{attribute 'qualified_only'}
VAR_GLOBAL
    
	MotorPosition  		AT %I* : UINT;
	CounterOverflow 	AT %I* : BOOL;
	CounterUnderflow 	AT %I* : BOOL;
	MotorEnable			AT %Q* : BOOL;
	MotorVelocity 		AT %Q* : INT;
	
END_VAR

(* stored: Version 1.1.0.1, ProductVersion 3.1.4024.9
   GVL GVL_Motor: Id {84b815ba-f4a9-4692-940e-12b636029e85} *)
